TYPE "UDT_HMI_Alarm_V2"
VERSION : 0.1
   STRUCT
      t : Struct
         x0 : Bool;
         x1 : Bool;
         x2 : Bool;
         x3 : Bool;
         x4 : Bool;
         x5 : Bool;
         x6 : Bool;
         x7 : Bool;
         x8 : Bool;
         x9 : Bool;
         x10 : Bool;
         x11 : Bool;
         x12 : Bool;
         x13 : Bool;
         x14 : Bool;
         x15 : Bool;
      END_STRUCT;
      iHmiSumAlm : Word;
   END_STRUCT;

END_TYPE

DATA_BLOCK "DeviceStatus_Alm"
{ S7_Optimized_Access := 'TRUE' }
VERSION : 0.1
NON_RETAIN
   VAR
      tEmergencyAlarm : Array["STARTARRAY".."DALARM"] of "UDT_HMI_Alarm_V2";   // stop machine fault
      tAlarm : Array["STARTARRAY".."DALARM"] of "UDT_HMI_Alarm_V2";   // stop next cycle faults
      tWarning : Array["STARTARRAY".."DALARM"] of "UDT_HMI_Alarm_V2";   // Generic warning
   END_VAR


BEGIN

END_DATA_BLOCK

DATA_BLOCK "DeviceStatus_Hmi"
{ S7_Optimized_Access := 'TRUE' }
VERSION : 0.1
NON_RETAIN
   VAR
      tHM_R : Struct
         tDevice : Array["STARTARRAY".."DEVICENUM_IND"] of Struct
            sName : String[20];
            iState : Int;   // (0=null;1=Not Conf,2=NotCon;3=Dis;4=Fault;5=Run)
         END_STRUCT;
      END_STRUCT;
      tHM_W : Struct
         b0 : Bool;
      END_STRUCT;
   END_VAR


BEGIN

END_DATA_BLOCK

